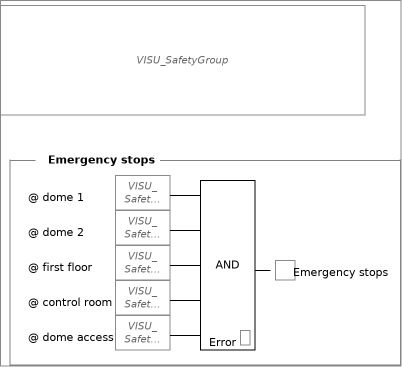
VISUALIZATION VISU_SafetyEmergencyStops  // 402x367
VAR_IN_OUT
	ref : SafetyEmergencyStops;
    widget : SafetyEmergencyStopsWidget;
END_VAR
    Polyline (160,160) (400,160) (400,365) (10,365) (10,160) (35,160)
    Label (45,150 110x20), "Emergency stops"
    Frame (115,175 55x35)
        shows VISU_SafetyEmergencyStop(contactNC := ref.dome1NC, contactNO := ref.dome1NO)
    Frame (115,245 55x35)
        shows VISU_SafetyEmergencyStop(contactNC := ref.firstFloorNC, contactNO := ref.firstFloorNO)
    Frame (115,280 55x35)
        shows VISU_SafetyEmergencyStop(contactNC := ref.controlRoomNC, contactNO := ref.controlRoomNO)
    Rectangle (200,180 55x170), "AND"
    Frame (240,330 10x15)
        shows VISU_State_green_red(state := ref.discrepancyError)
    Label (200,330 45x25), "Error"
    Label (25,185 80x25), "@ dome 1"
    Label (25,255 80x25), "@ first floor"
    Label (25,290 95x25), "@ control room"
    Line (255,270) (270,270), colour toggle: ref.allOK
    Frame (275,260 20x20)
        shows VISU_State_red_green(state := ref.allOK)
    Label (290,260 100x25), "Emergency stops"
    Frame (0,5 365x110)
        shows VISU_SafetyGroup(statusWidget := widget.actualStatus, comError := ref.groupComError, fbError := ref.groupFbError, outError := ref.groupOutError, reset := ref.processes.reset)
    Line (170,195) (200,195), colour toggle: ref.dome1NC
    Line (170,265) (200,265), colour toggle: ref.firstFloorNC
    Line (170,300) (200,300), colour toggle: ref.controlRoomNC
    Frame (115,210 55x35)
        shows VISU_SafetyEmergencyStop(contactNC := ref.dome2NC, contactNO := ref.dome2NO)
    Label (25,220 80x25), "@ dome 2"
    Line (170,230) (200,230), colour toggle: ref.dome2NC
    Frame (115,315 55x35)
        shows VISU_SafetyEmergencyStop(contactNC := ref.domeAccessNC, contactNO := ref.domeAccessNO)
    Label (25,325 95x25), "@ dome access"
    Line (170,335) (200,335), colour toggle: ref.domeAccessNC
END_VISUALIZATION

(* stored: Version 1.1.0.1, ProductVersion 3.1.4019.2
   Visu VISU_SafetyEmergencyStops: Id {5c3d6bb9-bf66-4a3c-9681-4e28ec2d22aa} *)
